FUNCTION_BLOCK Skill_FindLandmark6D EXTENDS FB_2_VisionSkills


VAR_INPUT
    // Vorhandene Eingänge beibehalten.

END_VAR

VAR_INPUT
    pQRCodeSkill : POINTER TO Skill_ReadQRCode;

    // Mandatory physical QR symbol edge length (not paper size).
    fQRCodeEdgeLengthMm : REAL;

    // Camera pose in robot-base coordinates at capture time.
    aRotation_BaseCamera    : TcVnMatrix3x3_LREAL;
    aTranslation_BaseCamera : TcVnVector3_LREAL;

    // Reject an unstable pose if the reprojection error exceeds this value.
    fMaxReprojectionErrorPx : LREAL := 2.0;

END_VAR

VAR_OUTPUT
    bLandmarkFound : BOOL;
    sLandmarkId    : STRING(255);

    // Full landmark pose in camera coordinates.
    aRotation_CameraLandmark    : TcVnMatrix3x3_LREAL;
    aTranslation_CameraLandmark : TcVnVector3_LREAL;

    // Full landmark pose in robot-base coordinates.
    aRotation_BaseLandmark    : TcVnMatrix3x3_LREAL;
    aTranslation_BaseLandmark : TcVnVector3_LREAL;

    // Quality and diagnosis.
    fReprojectionErrorPx : LREAL;
    hrLastError          : HRESULT;
END_VAR

VAR
    phase             : INT;
    l                 : INT;
    m                 : INT;
    k                 : INT;
    fHalfEdge         : REAL;
    aImagePoints      : ARRAY[0..3] OF TcVnPoint2_REAL;
    aReferencePoints  : ARRAY[0..3] OF TcVnPoint3_REAL;
    ipImagePoints     : ITcVnContainer;
    ipReferencePoints : ITcVnContainer;
    hr                : HRESULT;
    bStartedSubskill  : BOOL;
    bRunDone          : BOOL;
    fSum              : LREAL;
    resSubskill       : eResult;
	
	ipQRCodeContour : ITcVnContainer;
    aContourPoint   : TcVnPoint2_DINT;
END_VAR

CYCLIC_VISIONSKILL();

// Identity rotation matrix
aRotation_BaseCamera[0, 0] := 1.0;
aRotation_BaseCamera[0, 1] := 0.0;
aRotation_BaseCamera[0, 2] := 0.0;

aRotation_BaseCamera[1, 0] := 0.0;
aRotation_BaseCamera[1, 1] := 1.0;
aRotation_BaseCamera[1, 2] := 0.0;

aRotation_BaseCamera[2, 0] := 0.0;
aRotation_BaseCamera[2, 1] := 0.0;
aRotation_BaseCamera[2, 2] := 1.0;


// Zero translation vector
aTranslation_BaseCamera[0] := 0.0;
aTranslation_BaseCamera[1] := 0.0;
aTranslation_BaseCamera[2] := 200.0;



IF State = eState.Active THEN
    
	pQRCodeSkill^.Execute();
	
	IF pQRCodeSkill^.ExecutionDone AND pQRCodeSkill^.ExecutionResult = SUCCESS THEN
		sLandmarkId := pQRCodeSkill^.sCodeAsString;
		fHalfEdge := fQRCodeEdgeLengthMm * 0.5;

				// Get contour of first QR code.
		// ipCodeContourList is Vector<Vector<TcVnPoint2_DINT>>
		hr := F_VN_GetAt_ITcVnContainer(
			ipSrcContainer  := pQRCodeSkill^.ipCodeContourList,
			ipDestContainer := ipQRCodeContour,
			nIndex          := 0,
			hrPrev          := S_OK
		);
		
		// Extract the four QR corner points
		IF SUCCEEDED(hr) AND_THEN ipQRCodeContour <> 0 THEN
			FOR l := 0 TO 3 DO
				hr := F_VN_GetAt_TcVnPoint2_DINT(
					ipContainer := ipQRCodeContour,
					aElement    := aContourPoint,
					nIndex      := INT_TO_ULINT(l),
					hrPrev      := hr
				);
				IF SUCCEEDED(hr) THEN
					aImagePoints[l][0] := DINT_TO_REAL(aContourPoint[0]);
					aImagePoints[l][1] := DINT_TO_REAL(aContourPoint[1]);
				END_IF
			END_FOR
		
		END_IF

		// Known physical QR corners around the landmark origin.
		// Punkt 0: links oben beziehungsweise definierter Startpunkt
		aReferencePoints[0][0] := -fHalfEdge;
		aReferencePoints[0][1] := -fHalfEdge;
		aReferencePoints[0][2] := 0.0;
		
		// Punkt 1
		aReferencePoints[1][0] := fHalfEdge;
		aReferencePoints[1][1] := -fHalfEdge;
		aReferencePoints[1][2] := 0.0;
		
		// Punkt 2
		aReferencePoints[2][0] := fHalfEdge;
		aReferencePoints[2][1] := fHalfEdge;
		aReferencePoints[2][2] := 0.0;
		
		// Punkt 3
		aReferencePoints[3][0] := -fHalfEdge;
		aReferencePoints[3][1] := fHalfEdge;
		aReferencePoints[3][2] := 0.0;

		hr := F_VN_CreateContainer(
			ipImagePoints,
			ContainerType_Vector_TcVnPoint2_REAL,
			0,
			S_OK);
		
		hr := F_VN_CreateContainer(
			ipReferencePoints,
			ContainerType_Vector_TcVnPoint3_REAL,
			0,
			hr);
		
		FOR l := 0 TO 3 DO
			hr := F_VN_AppendToContainer_TcVnPoint2_REAL(
				aImagePoints[l],
				ipImagePoints,
				hr);
		
			hr := F_VN_AppendToContainer_TcVnPoint3_REAL(
				aReferencePoints[l],
				ipReferencePoints,
				hr);
		END_FOR
  
		hr := F_VN_SolvePnP(
			ipImagePoints           := ipImagePoints,
			ipReferencePoints       := ipReferencePoints,
			aCameraMatrix           := pOwnerCam^.aCameraMatrixLocal,
			aDistortionCoefficients := pOwnerCam^.aDistortionCoefficientsLocal,
			aRotationMatrix         := aRotation_CameraLandmark,
			aTranslationVector      := aTranslation_CameraLandmark,
			fReprojError            := fReprojectionErrorPx,
			hrPrev                  := S_OK);

		IF hr = S_OK THEN
			FOR l := 0 TO 2 DO
				FOR m := 0 TO 2 DO
					fSum := 0.0;
					FOR k := 0 TO 2 DO
						fSum := fSum
							+ aRotation_BaseCamera[l, k]
							* aRotation_CameraLandmark[k, m];
					END_FOR
					aRotation_BaseLandmark[l, m] := fSum;
				END_FOR
			END_FOR

			// t_B_L = R_B_C * t_C_L + t_B_C
			FOR l := 0 TO 2 DO
				fSum := aTranslation_BaseCamera[l];
				FOR k := 0 TO 2 DO
					fSum := fSum
						+ aRotation_BaseCamera[l, k]
						* aTranslation_CameraLandmark[k];
				END_FOR
				aTranslation_BaseLandmark[l] := fSum;
			END_FOR

		 bLandmarkFound := TRUE;
		 ExecutionDone:=TRUE;
		 ExecutionResult:=SUCCESS;
		 Deactivate();
   
		END_IF
		
	ELSIF pQRCodeSkill^.ExecutionDone AND pQRCodeSkill^.ExecutionResult = FAILURE THEN
		ExecutionDone:=TRUE;
		ExecutionResult:=FAILURE;
		Deactivate();
	END_IF
END_IF

METHOD PROTECTED OnActivate : eResult
VAR
    eParentResult : eResult;
    myResult      : eResult;
END_VAR

eParentResult := SUPER^.onActivate();
//--------------------------------------------------
myResult:=NONE;
// ----- YOUR CODE HERE (incl. Alarms) -------------
phase := 0;
bLandmarkFound := FALSE;
myResult:=SUCCESS;

// ----- END YOUR CODE -----------------------------
//--------------------------------------------------
onActivate := CombineResults(eParentResult,myResult);
END_METHOD

METHOD PROTECTED OnDeactivate : eResult
VAR
    eParentResult : eResult;
    myResult      : eResult;
END_VAR
eParentResult := SUPER^.onDeactivate();
//--------------------------------------------------
myResult:=NONE;
// ----- YOUR CODE HERE (incl. Alarms) -------------
phase := 0;
myResult:=SUCCESS;

// ----- END YOUR CODE -----------------------------
//--------------------------------------------------
onDeactivate := CombineResults(eParentResult,myResult);
END_METHOD

METHOD PROTECTED OnError : eResult
VAR
    eParentResult : eResult;
    myResult      : eResult;
END_VAR
eParentResult := SUPER^.onError();
//--------------------------------------------------
myResult:=NONE;
// ----- YOUR CODE HERE (incl. Alarms) -------------
ipImagePoints := 0;
ipReferencePoints := 0;
myResult:=SUCCESS;

// ----- END YOUR CODE -----------------------------
//--------------------------------------------------
onError := CombineResults(eParentResult, myResult);
END_METHOD

METHOD PROTECTED OnShutdown : eResult
VAR
    eParentResult : eResult;
    myResult      : eResult;
END_VAR
eParentResult := SUPER^.onShutdown();
//--------------------------------------------------
myResult:=NONE;
// ----- YOUR CODE HERE (incl. Alarms) -------------
phase := 0;
ipImagePoints := 0;
ipReferencePoints := 0;
myResult:=SUCCESS;

// ----- END YOUR CODE -----------------------------
//--------------------------------------------------
onShutdown := CombineResults(eParentResult, myResult);
END_METHOD

END_FUNCTION_BLOCK

(* stored: Version 1.1.0.1, ProductVersion 3.1.4026.18
   POU Skill_FindLandmark6D: Id {f74af431-203c-45ea-b1c5-99d698ba5355}, SpecialFunc None
   Folder StateControl: Id {f071cfd0-c82f-48d1-88d7-ad572fd8b5ec}
   Method OnActivate: Id {7a374fea-0c4d-40af-aaf4-06ebd09eb300}
   Method OnDeactivate: Id {22ccc076-a6b7-419c-a99d-0d58678c0ad4}
   Method OnError: Id {9a28fe08-923e-4c66-b184-a7131e6614b1}
   Method OnShutdown: Id {22712f1e-c3c0-49fd-b881-37948bb72a67} *)
